PROGRAM MAIN
VAR
	bTest_bool  AT %I* :  BOOL;
	iTest_int: INT;
	sTest_string: STRING;	
	DutTest: Dut_Test;
	fb_test: FB01;
END_VAR


sTest_String:='beckhoff';

bTest_bool:=TRUE;
DutTest.abc.a:=TRUE;
fb_test(input1:= , output1=> );

MotionGroup();

END_PROGRAM

(* stored: Version 1.1.0.1, ProductVersion 3.1.4024.11
   POU MAIN: Id {67c80a83-b5be-487e-bbb9-ca4534263da6}, SpecialFunc None *)
